Staubli VAL3: extractNum.pgx

public program extractNum(num& x_nInput[], num& x_nIndices[], num& x_nResult[])
  local num l_nElement
begin

  resize(x_nResult,1,size(x_nIndices))

  for l_nElement = 0 to size(x_nIndices)-1
    x_nResult[l_nElement] = x_nInput[x_nIndices[l_nElement]]
  endFor

end
